FUNCTION_BLOCK FB_PersistantDataStorage IMPLEMENTS I_PersistantDataStorage
VAR_INPUT
END_VAR
VAR_OUTPUT
END_VAR
VAR
END_VAR

END_FUNCTION_BLOCK

(* stored: Version 1.1.0.1
   POU FB_PersistantDataStorage: Id {9bee3f17-ef3d-4ebd-a47d-10e92d736a23}, SpecialFunc None *)
